(****************************************************************************************)
(*							Beckhoff Automation Poland									*)
(*								FB_SaveLineToFile  v2.0									*)
(*									26.06.2014											*)
(*						Blok funkcyjny zapisujacy tekst do pliku						*)
(*______________________________________________________________________________________
	Versions:
		v1.1	05.08.2016	* Przepisana wersja do TwinCat3
		v1.0	17.09.2012	* Podstawowa wersja z TwinCat2
________________________________________________________________________________________*)
FUNCTION_BLOCK FB_SaveLineToFile
VAR_INPUT
	bExecute	: BOOL;			(* Komenda wpisu *)
	AmsNetId	: T_AmsNetId;	(* AMS NET ID obiektu docelowego, gdy lokalnie, to zmienna moze byc pusta *)
	sPath		: STRING; 		(* Sciezka pliku, np  'Hard Disk\'*)
	sName		: STRING; 		(* Nazwa pliku wraz z rozszerzeniem 'LogFile.txt'; *)
	sLine		: STRING;		(* Tresc wpisu *)
END_VAR
VAR_OUTPUT
	bBusy		: BOOL;
	bError		: BOOL;
END_VAR
VAR
	fbFileOpen	: FB_FileOpen;
	ftOpen		: F_TRIG;
	fbFilePuts	: FB_FilePuts;
	ftPuts		: F_TRIG;
	fbFileClose	: FB_FileClose;
	ftClose		: F_TRIG;
END_VAR
VAR // added by the converter: edge detectors and wires of the graphical bodies
    _w1 : BOOL;
END_VAR

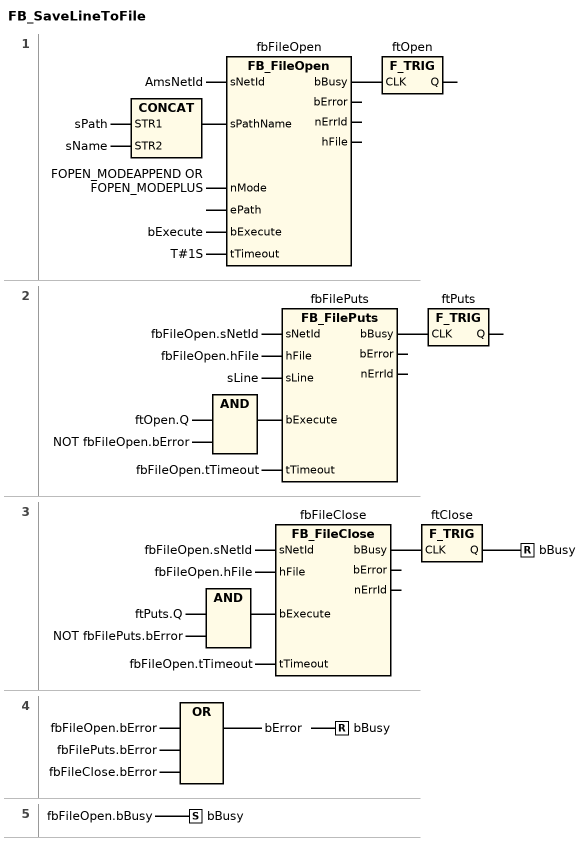
// NETWORK 1
fbFileOpen(
    sNetId := AmsNetId,
    sPathName := CONCAT(STR1 := sPath, STR2 := sName),
    nMode := FOPEN_MODEAPPEND OR FOPEN_MODEPLUS,
    bExecute := bExecute,
    tTimeout := T#1S); // FB_FileOpen
ftOpen(CLK := fbFileOpen.bBusy); // F_TRIG

// NETWORK 2
fbFilePuts(
    sNetId := fbFileOpen.sNetId,
    hFile := fbFileOpen.hFile,
    sLine := sLine,
    bExecute := ftOpen.Q AND (NOT fbFileOpen.bError),
    tTimeout := fbFileOpen.tTimeout); // FB_FilePuts
ftPuts(CLK := fbFilePuts.bBusy); // F_TRIG

// NETWORK 3
fbFileClose(
    sNetId := fbFileOpen.sNetId,
    hFile := fbFileOpen.hFile,
    bExecute := ftPuts.Q AND (NOT fbFilePuts.bError),
    tTimeout := fbFileOpen.tTimeout); // FB_FileClose
ftClose(CLK := fbFileClose.bBusy); // F_TRIG
bBusy R= ftClose.Q;

// NETWORK 4
_w1 := fbFileOpen.bError OR fbFilePuts.bError OR fbFileClose.bError;
bError := _w1;
bBusy R= _w1;

// NETWORK 5
bBusy S= fbFileOpen.bBusy;

END_FUNCTION_BLOCK

(* stored: Version 1.1.0.1, ProductVersion 3.1.4026.13, FileIdentifier 04e627c5a324fa1aaf8280fb8125b620ff9b9535, FileSignature 3947ef9f59edc47ebc14d938927d051703c1c5e4b4c9e09f894a248a91a4d2743856f6f81d36a48f3b0fa2b3a78cea30eaf8e4a13b32bb88711443380525ca12efb3066187e1e37dc89a644893ee63f790c3338d95d384ab072c4912f710183a4a604cdd1212817fcb998294b60d226879f4051cdea79bf0a5c578e42632393c07e9041190e7da916bd8bd0a159a74161754d705308b34322af39c496317e60c47829062bb9c4922f5f58934c48d4b0de0ce3e08806e4309099706f359f62fc66afde5a5a7a550a6ebe77bd81a8cf67e6905c23208c38bf7ff7733709c99a7359e46a94b6cc376c529199a7f2fd034a732a97b03754a446ffd563262e7b4498d
   POU FB_SaveLineToFile: Id {4b9bac5c-c356-411e-9365-203ea259bfc1}, SpecialFunc None *)
